FUNCTION read_bool_flag : BOOL
VAR_INPUT

	state : BOOL;
END_VAR
VAR
	ck0 : BOOL;
	ck1 : BOOL;
	ck2 : BOOL;
END_VAR

//Read bit register from Robot to PLC
ck0 := Robot_UR5.UR_outputs.B0;
ck1 := Robot_UR5.UR_outputs.B1;
ck2 := Robot_UR5.UR_outputs.B2;

IF (ck0=state AND ck1=state AND ck2=state) OR (ck0<>state AND ck1=state AND ck2=state) OR (ck0=state AND ck1<>state AND ck2=state) OR (ck0=state AND ck1=state AND ck2<>state) THEN
read_bool_flag := TRUE;
ELSE 
read_bool_flag := FALSE;	
END_IF

END_FUNCTION

(* stored: Version 1.1.0.1, ProductVersion 3.1.4024.4
   POU read_bool_flag: Id {4e9c11b2-cc43-48a5-a877-f4ce718a033a}, SpecialFunc None *)
